FUNCTION_BLOCK Stage19 (* Template for a Basic Function Block Type *)
  (* Standard: 61499-2 *)
  (* Version 1.0, 2021-06-20, HP *)
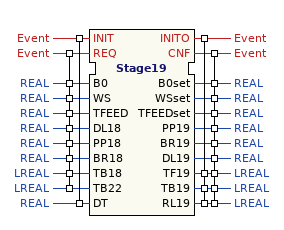
  EVENT_INPUT
    INIT WITH DT; (* Initialization Request *)
    REQ WITH B0, WS, TFEED, DL18, PP18, BR18, TB18, TB22; (* Normal Execution Request *)
  END_EVENT
  EVENT_OUTPUT
    INITO WITH TB19, RL19, TF19; (* Initialization Confirm *)
    CNF WITH TB19, DL19, TF19, BR19, PP19, RL19, B0set, WSset, TFEEDset; (* Execution Confirmation *)
  END_EVENT
  VAR_INPUT
    B0 : REAL;
    WS : REAL;
    TFEED : REAL;
    DL18 : REAL;
    PP18 : REAL;
    BR18 : REAL;
    TB18 : LREAL;
    TB22 : LREAL;
    DT : REAL;
  END_VAR
  VAR_OUTPUT
    B0set : REAL;
    WSset : REAL;
    TFEEDset : REAL;
    PP19 : REAL;
    BR19 : REAL;
    DL19 : REAL;
    TF19 : LREAL;
    TB19 : LREAL;
    RL19 : LREAL;
  END_VAR
  VAR
    AB : REAL; (* internal variabel *)
    UU : REAL;
    TREF : REAL;
    AD : REAL;
    AHC : REAL;
    AHR : REAL;
    AS : REAL;
    REC : REAL;
    WN : REAL;
    WN_1 : REAL;
    XKN : REAL;
    C1 : REAL;
    HS : REAL;
    G : REAL;
    W1 : REAL;
    TFREC : REAL;
    TS : REAL;
    DTS : REAL;
    TF19_last : REAL;
    RL19_last : REAL;
    TB19_last : REAL;
    USS : REAL;
    RHOB : REAL;
    CPB : REAL;
    CPF : REAL;
    FMW : REAL;
    HLV : REAL;
    HV : REAL;
    BPR : REAL;
    FMC : REAL;
    U : REAL;
    A : REAL;
    B : REAL;
    C : REAL;
    D1 : REAL;
    d : REAL;
    a : REAL;
    A1 : REAL;
    A2 : REAL;
    A3 : REAL;
    A4 : REAL;
    A5 : REAL;
    A6 : REAL;
    p : REAL;
    q : REAL;
    TC : REAL;
    PC : REAL;
    DTB19 : REAL;
    DEN19 : REAL;
    DH19 : REAL;
    DP19 : REAL;
    DPDH19 : REAL;
    DT19 : REAL;
    m : REAL;
    n : REAL;
    VR19 : REAL;
    DELTA19 : REAL;
    DELTA41 : REAL;
    DELTA63 : REAL;
    DELTA19_last : REAL;
    DELTA41_last : REAL;
    DELTA63_last : REAL;
  END_VAR
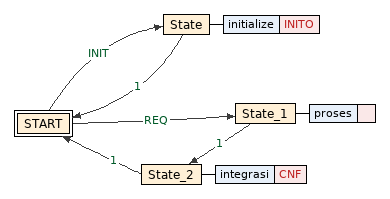
  EC_STATES
    START; (* Initial State *)
    State : initialize -> INITO;
    State_1 : proses;
    State_2 : integrasi -> CNF;
  END_STATES
  EC_TRANSITIONS
    START TO State := INIT;
    State TO START := 1;
    START TO State_1 := REQ;
    State_1 TO State_2 := 1;
    State_2 TO START := 1;
  END_TRANSITIONS
  ALGORITHM initialize IN ST: (* Initialization algorithm *)
TREF :=273.15;
AB :=57.2727;
AHC :=4069.2;
AHR :=2639.7;
AS :=3225.7;
REC :=0.0;
//TF2:=TF2;

//TFEED :=TFEED1+TREF;
 //TS:=TS1+TREF;
WN :=3.0;
XKN :=0.68;
HS:=0.11;
G :=9.81;
W1 :=0.50;

RL19 := 0.621148983552414;
TB19 := 319.429927458879;
TB22:=314.548634310388;
TF19 := 316.357381861072;




RL19_last :=RL19;
TB19_last :=TB19;
TF19_last :=TF19;
  END_ALGORITHM
  ALGORITHM proses IN ST: (* kalkulasi *)
UU := TFEED;
TFREC:=TB22;
U :=UU;

USS :=49.767;
C1 :=0.625;
RHOB :=1032.4; //maassa jenis brine
CPB :=1.00; //heatcapacity Brine
CPF :=1.00; //heat capacity feed
FMW :=23654.0;
HLV :=563.7959;
HV :=625.1971;
BPR :=2.192;
FMC :=34736.09;
//U :=UU; //feed temp



///  Calculate the physical properties

//A :=3.2437814;
//B :=5.86826*0.001;
//C :=1.1702379*0.00000001;
//D1 :=2.1878462*0.001;
//TC :=647.27;
//PC :=218.167;


A1 :=3.2437814;
A2:=5.86826*0.001;
A3:=1.1702379*0.00000001;
A4 :=2.1878462*0.001;
A5 :=647.27;
A6 :=218.167;

DTB19 :=A5-TB19;
DEN19 :=(A1+A2*DTB19+A3*DTB19*DTB19*DTB19)/(1+A4*DTB19)*DTB19/TB19;
p:=DEN19;
q:=10.0;
PP19 :=A6/(EXPT(q, p));

// calculate the brine flow rates
DP19:=PP18-PP19;
DH19:=RL19-C1*HS;
DPDH19 :=DP19*101000+G*RHOB*DH19;
m:=DPDH19*RHOB;
n:=0.5;
BR19 :=WN*XKN*RL19*(EXPT(m, n));
BR19 :=BR19*60.0/1000.0;

// calculate the vapor flow rates

DT19 :=TB19-BPR/1.8-(TFREC+TF19)*0.5;
VR19:=U*AHC*DT19/HLV/1000.0;
DL19 :=DL18+VR19;


//// state equation
DELTA19 :=(BR18-BR19-VR19)*1000.0/RHOB/AB;
DELTA41 :=((BR18*CPB*(TB18-TB19))-VR19*(HV-CPB*(TB19-TREF)))*1000.0/AB/RHOB/CPB/RL19;
DELTA63 :=(B0*CPF*(TFREC-TF19)*1000+(U*AHC*DT19))/FMW/CPF;
;
  END_ALGORITHM
  ALGORITHM integrasi IN ST: (* new algorithm *)
B0set:=B0;
WSset:=WS ;
TFEEDset:=TFEED;
//integrasi
RL19 := (DELTA19 + DELTA19_last)*0.5*DT + RL19_last;
DELTA19_last :=DELTA19 ;
RL19_last :=RL19;

TB19:= (DELTA41 + DELTA41_last)*0.5*DT + TB19_last;
DELTA41_last :=DELTA41 ;
TB19_last:=TB19;

TF19 := (DELTA63 + DELTA63_last)*0.5*DT + TF19_last;
DELTA63_last :=DELTA63 ;
TF19_last :=TF19;
  END_ALGORITHM
END_FUNCTION_BLOCK
